VAR_GLOBAL
	Eixo1 : AXIS_REF;
	Eixo2 : AXIS_REF;
END_VAR

(* stored: Version 1.1.0.1, ProductVersion 3.1.4024.13
   GVL Eixos: Id {cd822f58-4ec7-4654-884b-94451a9a0046} *)
